FUNCTION_BLOCK IX (* Service Interface Function Block Type *)
  (* Standard: 61499-2 *)
  (* Version 0.0, 2014-08-26, 4DIAC-IDE, 4DIAC-Consortium *)
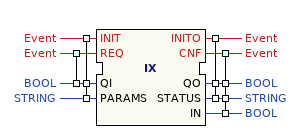
  EVENT_INPUT
    INIT WITH QI, PARAMS; (* Service Initialization *)
    REQ WITH QI; (* Service Request *)
  END_EVENT
  EVENT_OUTPUT
    INITO WITH QO, STATUS; (* Initialization Confirm *)
    CNF WITH QO, STATUS, IN; (* Confirmation of Requested Service *)
  END_EVENT
  VAR_INPUT
    QI : BOOL; (* Event Input Qualifier *)
    PARAMS : STRING; (* Service Parameters *)
  END_VAR
  VAR_OUTPUT
    QO : BOOL; (* Event Output Qualifier *)
    STATUS : STRING; (* Service Status *)
    IN : BOOL; (* Input data from resource *)
  END_VAR
  SERVICE APPLICATION/RESOURCE (* Service Interface Function Block Type *)
    SEQUENCE normal_establishment
      APPLICATION.INIT+(PARAMS) -> APPLICATION.INITO+(PARAMS);
    END_SEQUENCE
    SEQUENCE unsuccessful_establishment
      APPLICATION.INIT+(PARAMS) -> APPLICATION.INITO-(STATUS);
    END_SEQUENCE
    SEQUENCE request_confirm
      APPLICATION.REQ+(SD) -> APPLICATION.CNF+(RD);
    END_SEQUENCE
    SEQUENCE request_inhibited
      APPLICATION.REQ-(SD) -> APPLICATION.CNF-(STATUS);
    END_SEQUENCE
    SEQUENCE request_error
      APPLICATION.REQ+(SD) -> APPLICATION.CNF-(STATUS);
    END_SEQUENCE
    SEQUENCE indication_response
      RESOURCE.indicate(RD) -> APPLICATION.IND+(RD);
      APPLICATION.RSP(QI,SD) -> RESOURCE.response(QI,SD);
    END_SEQUENCE
    SEQUENCE indication_inhibited
      RESOURCE.indicate(RD,QI=FALSE) -> RESOURCE.inhibited();
    END_SEQUENCE
    SEQUENCE error_indication
      RESOURCE.error(STATUS) -> APPLICATION.IND-(STATUS);
    END_SEQUENCE
    SEQUENCE application_initiated_termination
      APPLICATION.INIT-() -> APPLICATION.INITO-(STATUS);
    END_SEQUENCE
    SEQUENCE resource_initiated_termination
      -> APPLICATION.INITO-(STATUS);
    END_SEQUENCE
  END_SERVICE
END_FUNCTION_BLOCK
